// TIA Portal V19 export
TYPE "PARAMETERADDR"
   STRUCT
      ATTRIBUTE : Byte;
      NO_ELEM : Byte;
      PARA_NO : Word;
      SUBINDEX : Word;
   END_STRUCT;
END_TYPE
